% RSLogix 500 project P7_KOBIERSKI_M_v2.RSS, saved by version 8.30.00.16 %
PROJECT "UNTITLED"    % processor: Bul.1763 MicroLogix 1100 Series B %

PROGRAM FILES
  LAD 2 "MAIN"  6 rungs
  LAD 3 "IO"  5 rungs
  LAD 4 "CYCLE"  2 rungs
  LAD 5 "CTRL"  3 rungs
  LAD 6 "CALIB"  9 rungs
  LAD 7 "SIM"  4 rungs

DATA FILES
  O0 OUTPUT  4 elements
  I1 INPUT  6 elements
  S2 STATUS  66 elements
  B3 BINARY  1 elements
  T4 TIMER  4 elements
  C5 COUNTER  2 elements
  R6 CONTROL  1 elements
  N7 INTEGER  8 elements
  F8 FLOAT  10 elements
  N9 SIM VALUES  3 elements

LADDER 2 "MAIN"
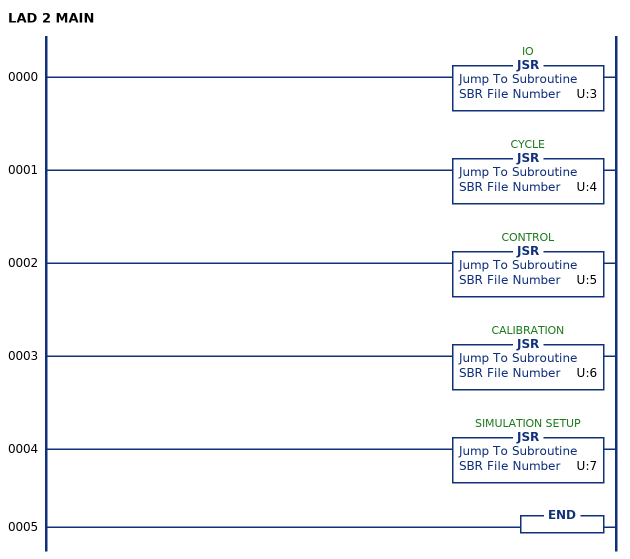
% Rung: 0 %
SOR JSR U:3 EOR
%   U:3  "IO" %
% Rung: 1 %
SOR JSR U:4 EOR
%   U:4  "CYCLE" %
% Rung: 2 %
SOR JSR U:5 EOR
%   U:5  "CONTROL" %
% Rung: 3 %
SOR JSR U:6 EOR
%   U:6  "CALIBRATION" %
% Rung: 4 %
SOR JSR U:7 EOR
%   U:7  "SIMULATION SETUP" %
% Rung: 5 %
SOR END EOR

LADDER 3 "IO"
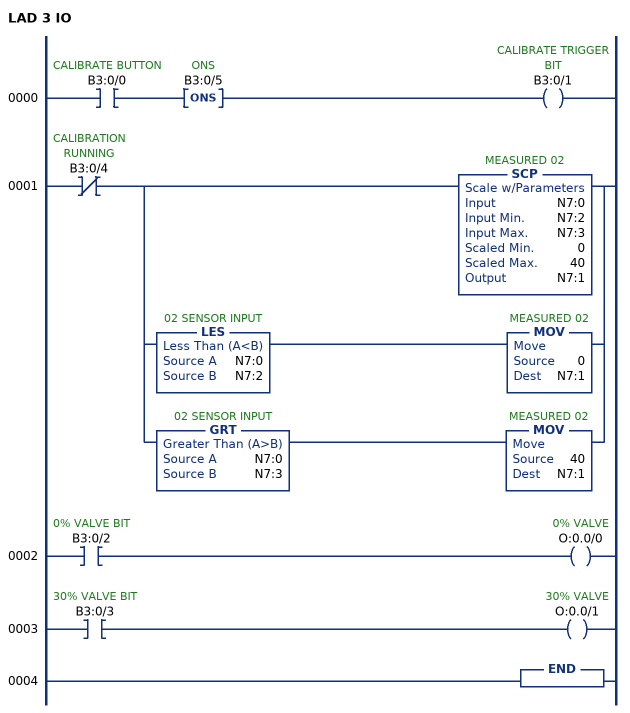
% Rung: 0 %
SOR XIC B3:0/0 ONS B3:0/5 OTE B3:0/1 EOR
%   B3:0/0  "CALIBRATE BUTTON" %
%   B3:0/5  "ONS" %
%   B3:0/1  "CALIBRATE TRIGGER BIT" %
% Rung: 1 %
SOR XIO B3:0/4 BST SCP N7:0 N7:2 N7:3 0 40 N7:1 NXB LES N7:0 N7:2 MOV 0 N7:1 NXB GRT N7:0 N7:3 MOV 40 N7:1 BND EOR
%   B3:0/4  "CALIBRATION RUNNING" %
%   N7:0  "02 SENSOR INPUT" %
%   N7:2  "02 INPUT MIN" %
%   N7:3  "02 INPUT MAX" %
%   N7:1  "MEASURED 02" %
% Rung: 2 %
SOR XIC B3:0/2 OTE O:0.0/0 EOR
%   B3:0/2  "0% VALVE BIT" %
%   O:0.0/0  "0% VALVE" %
% Rung: 3 %
SOR XIC B3:0/3 OTE O:0.0/1 EOR
%   B3:0/3  "30% VALVE BIT" %
%   O:0.0/1  "30% VALVE" %
% Rung: 4 %
SOR END EOR

LADDER 4 "CYCLE"
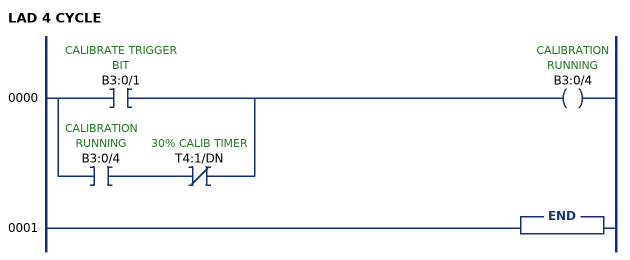
% Rung: 0 %
SOR BST XIC B3:0/1 NXB XIC B3:0/4 XIO T4:1/DN BND OTE B3:0/4 EOR
%   B3:0/1  "CALIBRATE TRIGGER BIT" %
%   B3:0/4  "CALIBRATION RUNNING" %
%   T4:1  "30% CALIB TIMER" %
% Rung: 1 %
SOR END EOR

LADDER 5 "CTRL"
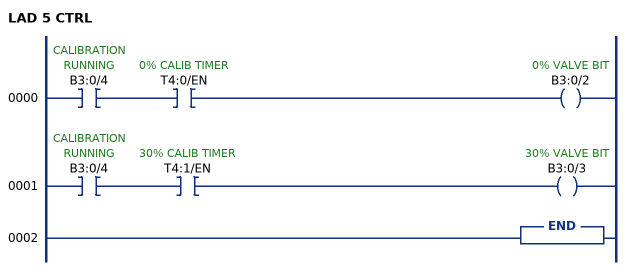
% Rung: 0 %
SOR XIC B3:0/4 XIC T4:0/EN OTE B3:0/2 EOR
%   B3:0/4  "CALIBRATION RUNNING" %
%   T4:0  "0% CALIB TIMER" %
%   B3:0/2  "0% VALVE BIT" %
% Rung: 1 %
SOR XIC B3:0/4 XIC T4:1/EN OTE B3:0/3 EOR
%   B3:0/4  "CALIBRATION RUNNING" %
%   T4:1  "30% CALIB TIMER" %
%   B3:0/3  "30% VALVE BIT" %
% Rung: 2 %
SOR END EOR

LADDER 6 "CALIB"
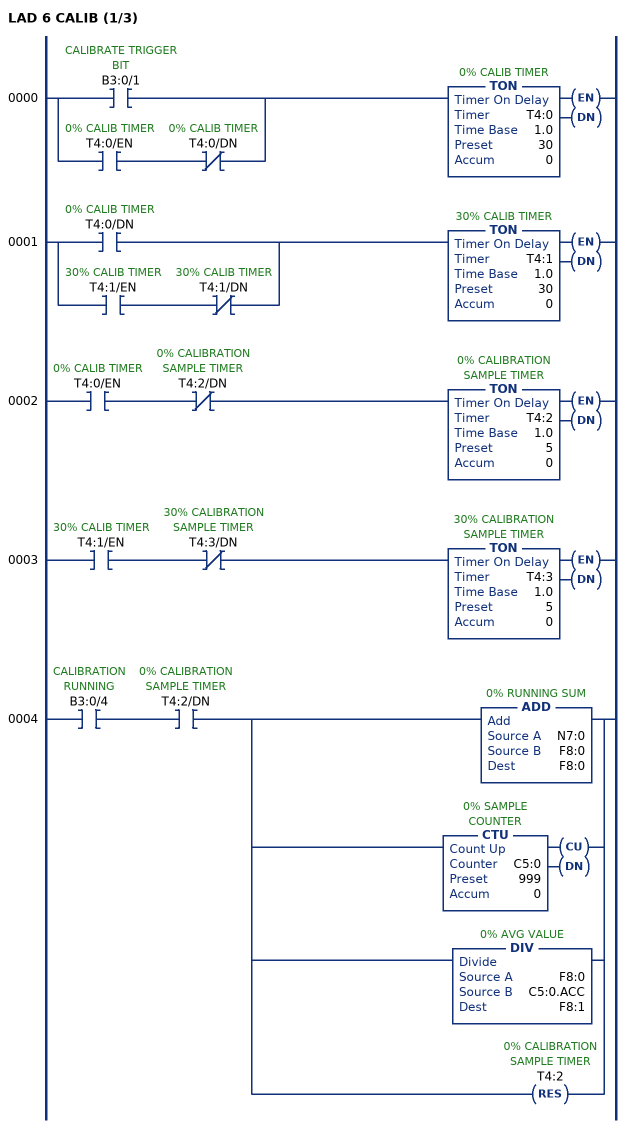
% Rung: 0 %
SOR BST XIC B3:0/1 NXB XIC T4:0/EN XIO T4:0/DN BND TON T4:0 1.0 30 0 EOR
%   B3:0/1  "CALIBRATE TRIGGER BIT" %
%   T4:0  "0% CALIB TIMER" %
% Rung: 1 %
SOR BST XIC T4:0/DN NXB XIC T4:1/EN XIO T4:1/DN BND TON T4:1 1.0 30 0 EOR
%   T4:0  "0% CALIB TIMER" %
%   T4:1  "30% CALIB TIMER" %
% Rung: 2 %
SOR XIC T4:0/EN XIO T4:2/DN TON T4:2 1.0 5 0 EOR
%   T4:0  "0% CALIB TIMER" %
%   T4:2  "0% CALIBRATION SAMPLE TIMER" %
% Rung: 3 %
SOR XIC T4:1/EN XIO T4:3/DN TON T4:3 1.0 5 0 EOR
%   T4:1  "30% CALIB TIMER" %
%   T4:3  "30% CALIBRATION SAMPLE TIMER" %
% Rung: 4 %
SOR XIC B3:0/4 XIC T4:2/DN BST ADD N7:0 F8:0 F8:0 NXB CTU C5:0 999 0 NXB DIV F8:0 C5:0.ACC F8:1 NXB RES T4:2 BND EOR
%   B3:0/4  "CALIBRATION RUNNING" %
%   T4:2  "0% CALIBRATION SAMPLE TIMER" %
%   N7:0  "02 SENSOR INPUT" %
%   F8:0  "0% RUNNING SUM" %
%   C5:0  "0% SAMPLE COUNTER" %
%   F8:1  "0% AVG VALUE" %

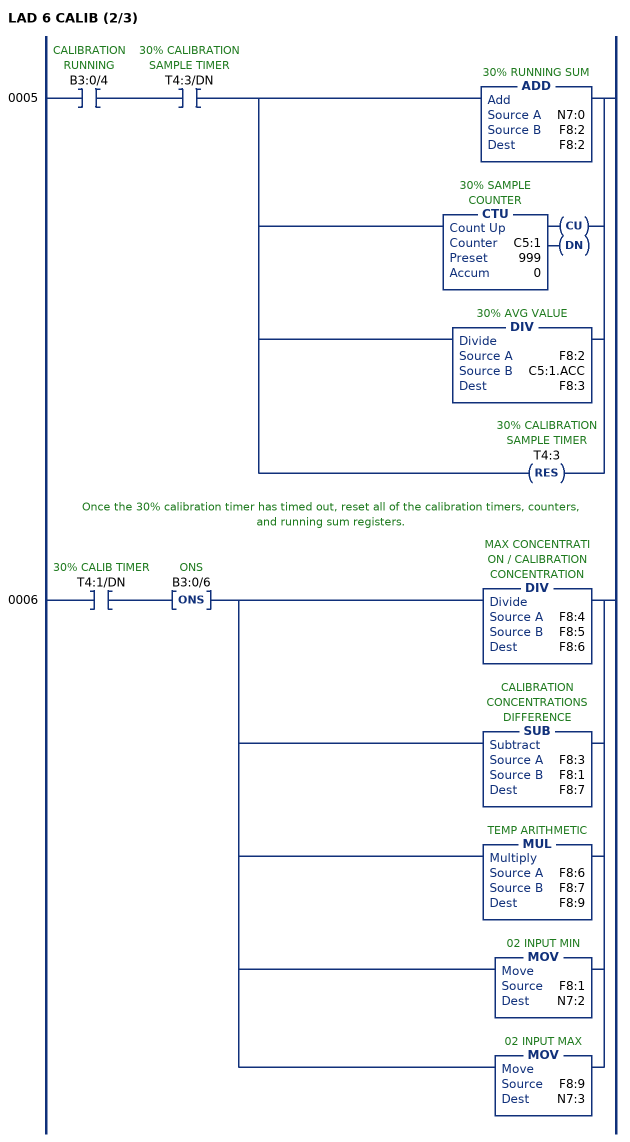
% Rung: 5 %
SOR XIC B3:0/4 XIC T4:3/DN BST ADD N7:0 F8:2 F8:2 NXB CTU C5:1 999 0 NXB DIV F8:2 C5:1.ACC F8:3 NXB RES T4:3 BND EOR
%   B3:0/4  "CALIBRATION RUNNING" %
%   T4:3  "30% CALIBRATION SAMPLE TIMER" %
%   N7:0  "02 SENSOR INPUT" %
%   F8:2  "30% RUNNING SUM" %
%   C5:1  "30% SAMPLE COUNTER" %
%   F8:3  "30% AVG VALUE" %
% Rung: 6 %
% Once the 30% calibration timer has timed out, reset all of the calibration timers, counters, and running sum registers. %
SOR XIC T4:1/DN ONS B3:0/6 BST DIV F8:4 F8:5 F8:6 NXB SUB F8:3 F8:1 F8:7 NXB MUL F8:6 F8:7 F8:9 NXB MOV F8:1 N7:2 NXB MOV F8:9 N7:3 BND EOR
%   T4:1  "30% CALIB TIMER" %
%   B3:0/6  "ONS" %
%   F8:4  "SENSOR MAX CONCENTRATION" %
%   F8:5  "30% CALIBRATION GAS CONCENTRATION" %
%   F8:6  "MAX CONCENTRATION / CALIBRATION CONCENTRATION" %
%   F8:3  "30% AVG VALUE" %
%   F8:1  "0% AVG VALUE" %
%   F8:7  "CALIBRATION CONCENTRATIONS DIFFERENCE" %
%   F8:9  "TEMP ARITHMETIC" %
%   N7:2  "02 INPUT MIN" %
%   N7:3  "02 INPUT MAX" %

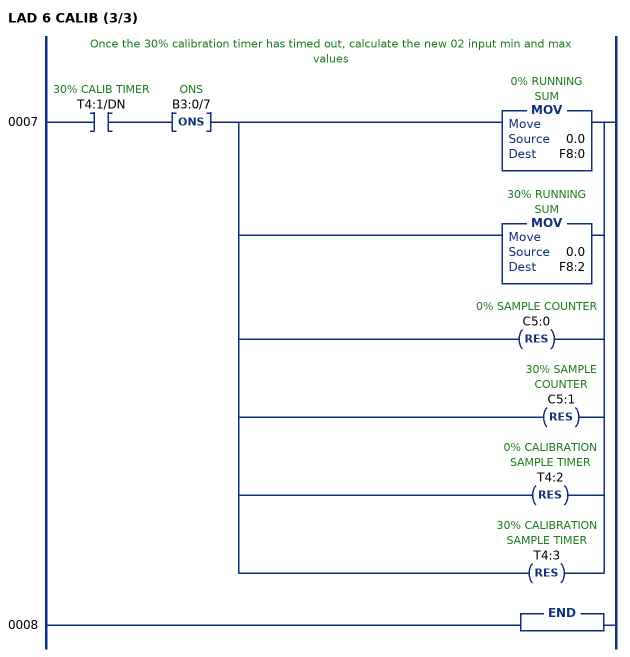
% Rung: 7 %
% Once the 30% calibration timer has timed out, calculate the new 02 input min and max values %
SOR XIC T4:1/DN ONS B3:0/7 BST MOV 0.0 F8:0 NXB MOV 0.0 F8:2 NXB RES C5:0 NXB RES C5:1 NXB RES T4:2 NXB RES T4:3 BND EOR
%   T4:1  "30% CALIB TIMER" %
%   B3:0/7  "ONS" %
%   F8:0  "0% RUNNING SUM" %
%   F8:2  "30% RUNNING SUM" %
%   C5:0  "0% SAMPLE COUNTER" %
%   C5:1  "30% SAMPLE COUNTER" %
%   T4:2  "0% CALIBRATION SAMPLE TIMER" %
%   T4:3  "30% CALIBRATION SAMPLE TIMER" %
% Rung: 8 %
SOR END EOR

LADDER 7 "SIM"
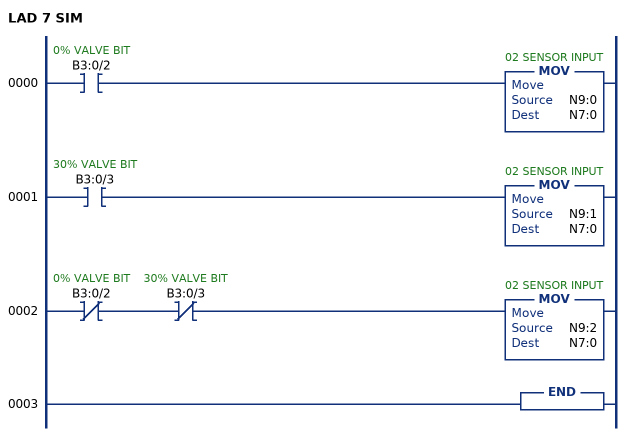
% Rung: 0 %
SOR XIC B3:0/2 MOV N9:0 N7:0 EOR
%   B3:0/2  "0% VALVE BIT" %
%   N9:0  "SIMULATED 0% INPUT INT" %
%   N7:0  "02 SENSOR INPUT" %
% Rung: 1 %
SOR XIC B3:0/3 MOV N9:1 N7:0 EOR
%   B3:0/3  "30% VALVE BIT" %
%   N9:1  "SIMULATED 30% INPUT INT" %
%   N7:0  "02 SENSOR INPUT" %
% Rung: 2 %
SOR XIO B3:0/2 XIO B3:0/3 MOV N9:2 N7:0 EOR
%   B3:0/2  "0% VALVE BIT" %
%   B3:0/3  "30% VALVE BIT" %
%   N9:2  "SIMULATED OPERATING INPUT INT" %
%   N7:0  "02 SENSOR INPUT" %
% Rung: 3 %
SOR END EOR

DATA TABLE (non-zero values as saved)
DATA T4
% .PRE .ACC %
% T4:0 % 30 0
% T4:1 % 30 0
% T4:2 % 5 0
% T4:3 % 5 0
DATA C5
% .PRE .ACC %
% C5:0 % 999 0
% C5:1 % 999 0
DATA N7
% N7:0 % 0 0 0 16383 0 0 0 0
DATA F8
% F8:0 % 0 0 0 0 40
% F8:5 % 30 0 0 0 0
DATA N9
% N9:0 % 0 12288 8192
